FUNCTION_BLOCK FB_AxisWriteNC
VAR_INPUT
	bExecute: BOOL;
	bReset: BOOL;
END_VAR
VAR_IN_OUT
	stConfig: ST_AxisParams;
	Axis: AXIS_REF;
END_VAR
VAR_OUTPUT
	bDone: BOOL;
	bBusy: BOOL;
	bError: BOOL;
	nErrorID: UDINT;
END_VAR
VAR
{% for item in nc_params %}
  {% if item.is_bool %}
	{{ item.fb_write }}: MC_WriteBoolParameter;
  {% else %}
	{{ item.fb_write }}: MC_WriteParameter;
  {% endif %}
{% endfor %}
END_VAR

// File auto-generated! Take care editing!
// Clears errors and allows a new read
IF bReset THEN
	bExecute := FALSE;
	bReset := FALSE;
END_IF
{% for item in nc_params %}
{{ item.fb_write }}(Execute:=bExecute,
	ParameterNumber:=MC_AxisParameter.{{ item.MC_AxisParameter }},
	Value:=stConfig.{{ item.stConfig }},
	Axis:=Axis);
{% endfor %}
bDone := {{ nc_params|join(' AND ', attribute='fb_write_done') }};
bBusy := {{ nc_params|join(' OR ', attribute='fb_write_busy') }};
bError := {{ nc_params|join(' OR ', attribute='fb_write_error') }};
IF NOT bError THEN
	nErrorID := 0;
{% for item in nc_params %}
ELSIF {{ item.fb_write }}.ErrorID > 0 THEN
	nErrorID := {{ item.fb_write }}.ErrorID;
{% endfor %}
END_IF

END_FUNCTION_BLOCK

(* stored: Version 1.1.0.1, ProductVersion 3.1.4020.12
   POU FB_AxisWriteNC: Id {f7f47c17-7b1c-42c7-9653-657995f4107e}, SpecialFunc None *)
